SYSTEM ASM_VIEWL (* Assembly Station with Dual Stroke Cylinder *)
  (* Standard: 61499-1; Classification: Simulation; ApplicationDomain: Assembly; Type: Dual Stroke Cylinder *)
  (* Version 0.0, 2003-03-15, JHC, Rockwell Automation, Adapted from DRILL_VIEWL *)
  DEVICE HMI : FRAME_DEVICE
    RESOURCE RES1 : PANEL_RESOURCE
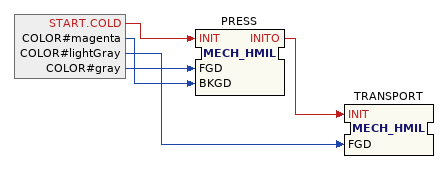
      FBS
        PRESS : MECH_HMIL;
        TRANSPORT : MECH_HMIL;
      END_FBS
      EVENT_CONNECTIONS
        START.COLD TO PRESS.INIT;
        PRESS.INITO TO TRANSPORT.INIT;
      END_CONNECTIONS
      DATA_CONNECTIONS
        COLOR#magenta TO PRESS.FGD;
        COLOR#lightGray TO TRANSPORT.FGD;
        COLOR#gray TO PRESS.BKGD;
      END_CONNECTIONS
    END_RESOURCE
  END_DEVICE
  DEVICE VIEW : FRAME_DEVICE
    RESOURCE ASSEMBLY : VIEW_PANEL
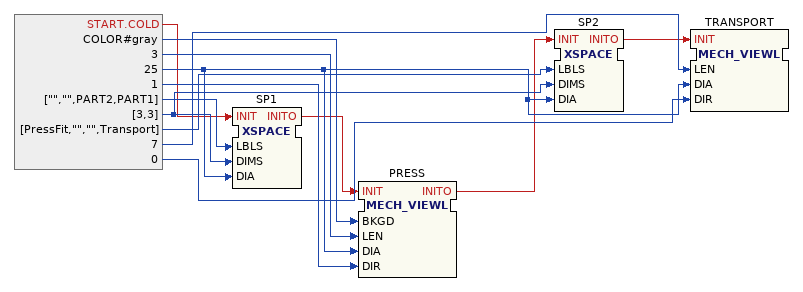
      FBS
        SP1 : XSPACE;
        PRESS : MECH_VIEWL; (* Vertical press element *)
        SP2 : XSPACE;
        TRANSPORT : MECH_VIEWL; (* Horizontal transport (dual-stroke cylinder) *)
      END_FBS
      EVENT_CONNECTIONS
        START.COLD TO SP1.INIT;
        SP1.INITO TO PRESS.INIT;
        PRESS.INITO TO SP2.INIT;
        SP2.INITO TO TRANSPORT.INIT;
      END_CONNECTIONS
      DATA_CONNECTIONS
        COLOR#gray TO PRESS.BKGD;
        3 TO PRESS.LEN;
        25 TO PRESS.DIA;
        1 TO PRESS.DIR;
        ["","",PART2,PART1] TO SP1.LBLS;
        [3,3] TO SP1.DIMS;
        25 TO SP1.DIA;
        [PressFit,"","",Transport] TO SP2.LBLS;
        [3,3] TO SP2.DIMS;
        25 TO SP2.DIA;
        7 TO TRANSPORT.LEN;
        25 TO TRANSPORT.DIA;
        0 TO TRANSPORT.DIR;
      END_CONNECTIONS
    END_RESOURCE
    DATA_CONNECTIONS
      0 TO ASSEMBLY.TRACE;
      25 TO ASSEMBLY.DIA;
      [7,5] TO ASSEMBLY.SIZE;
      0 TO ASSEMBLY.VERTICAL;
    END_CONNECTIONS
  END_DEVICE
  DATA_CONNECTIONS (* parameter values *)
    [100,100,380,100] TO HMI.BOUNDS;
    [1,1] TO HMI.GRID;
    [480,100,185,150] TO VIEW.BOUNDS;
  END_CONNECTIONS
END_SYSTEM
